(* PLC project Unnamed, Unknown Unnamed 1 *)
(* stored: creationDateTime 2019-04-18T11:44:44, modificationDateTime 2021-02-08T14:39:08 *)

PROGRAM Hello_World
  VAR
    level AT %IW101 : UINT;
    outflow AT %QW100 : UINT;
  END_VAR
  VAR
    max_level : REAL := 1200.0;
    min_level : REAL := 800.0;
    convert_to_level : REAL := 32.768;  (* Convert from u16 modbus to real level value in mm *)
    convert_from_flow : REAL := 1638.4;  (* Convert from real outflow value to u16 modbus *)
    low_flow : REAL := 15.0;  (* Low flow *)
    high_flow : REAL := 25.0;  (* high flow *)
  END_VAR
  VAR  (* added by the conversion: wires and edge detectors of the diagram *)
    _DIV10_OUT : REAL;
    _SEL15_OUT : ANY;
  END_VAR

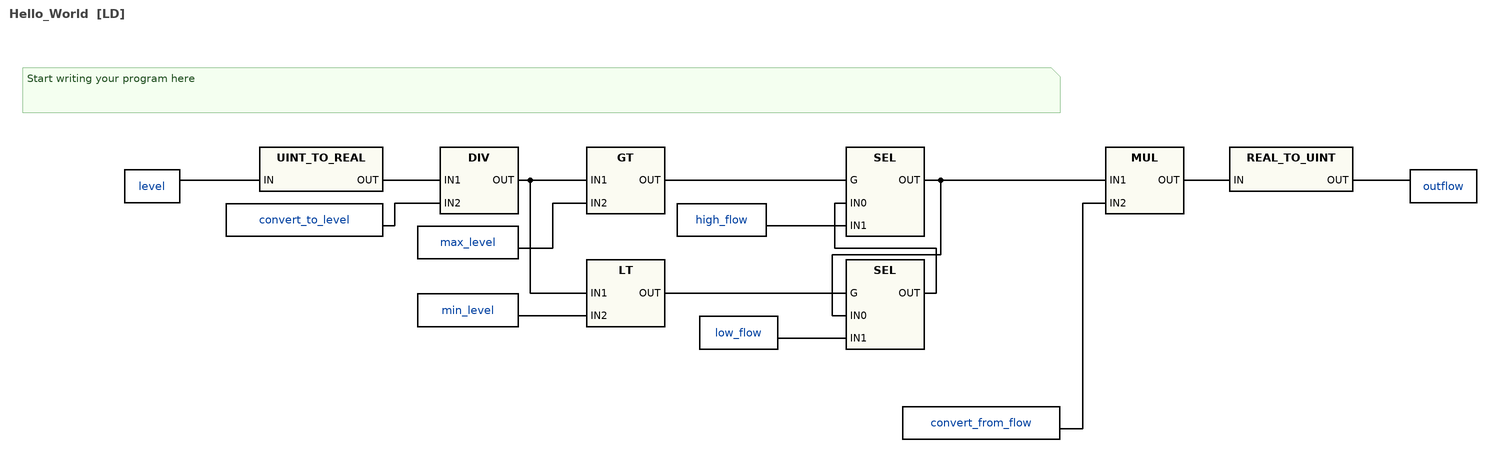
(* LD diagram, written out as Structured Text *)
(* Start writing your program here *)
_DIV10_OUT := UINT_TO_REAL(level) / convert_to_level;
_SEL15_OUT := SEL(_DIV10_OUT > max_level, SEL(_DIV10_OUT < min_level, _SEL15_OUT, low_flow), high_flow);
outflow := REAL_TO_UINT(_SEL15_OUT * convert_from_flow);
END_PROGRAM

CONFIGURATION Config0
  RESOURCE Res0 ON PLC
    TASK task0(INTERVAL := T#300ms, PRIORITY := 0);
    PROGRAM instance0 WITH task0 : Hello_World;
  END_RESOURCE
END_CONFIGURATION
